FUNCTION_BLOCK Valve_Digital
VAR_INPUT
	//Open Feedback from Valve
	Open_Feedback : BOOL; 
	//Closed Feedback from Valve
	Closed_Feedback : BOOL;
	//Open Request from PLC Program
	Open_Request : BOOL;
	//Triggered from alarm ladder
	Fail_to_Open : BOOL;
	//Triggered from Alarm ladder
	Fail_to_Close : BOOL;
END_VAR
VAR_OUTPUT
	//Tells the valve to open when true, close when False
	Open_Command : BOOL;
END_VAR
VAR	
END_VAR

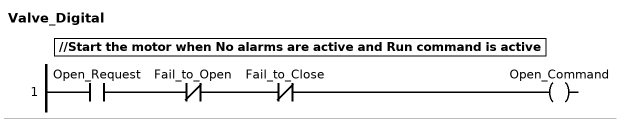
// NETWORK 1
// label: //Start the motor when No alarms are active and Run command is active
Open_Command := Open_Request AND NOT Fail_to_Open AND NOT Fail_to_Close;

END_FUNCTION_BLOCK

(* stored: Version 1.1.0.1, ProductVersion 3.1.4024.12
   POU Valve_Digital: Id {98e771d8-3fe1-4057-aa61-fd7121110cde}, SpecialFunc None *)
